PROGRAM MAIN
VAR
END_VAR

END_PROGRAM

(* stored: Version 1.1.0.1
   POU MAIN: Id {0a491740-e92b-4959-a911-54da94aeaf18} *)
